// Mitsubishi GX Works2 project: pr2   PLC: Q03UDV

PROGRAM MAIN
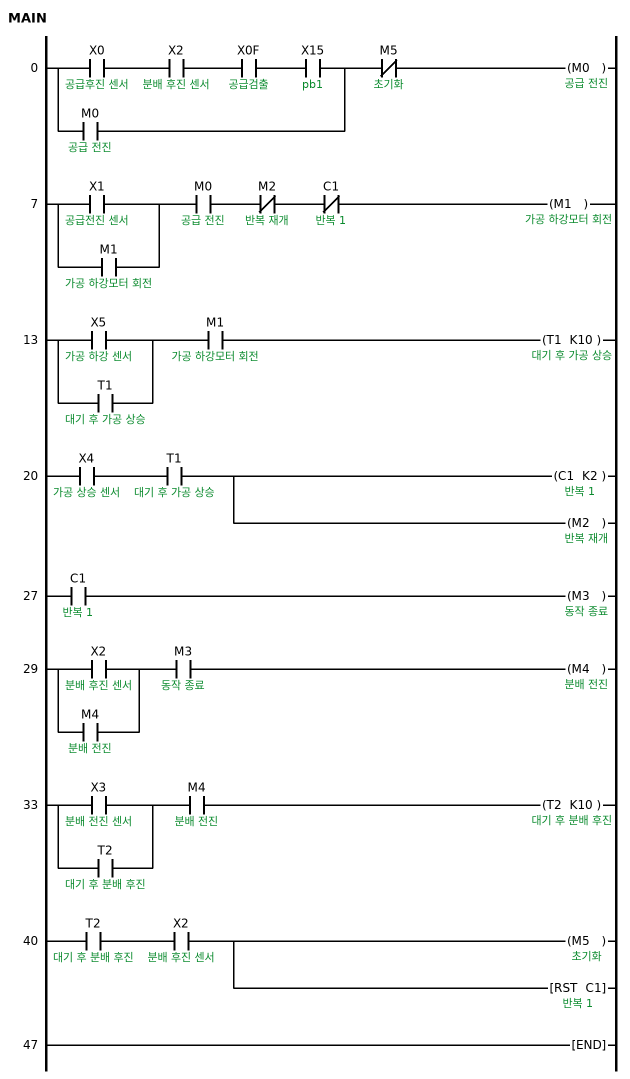
0     LD      X0  ; 공급후진 센서
      AND     X2  ; 분배 후진 센서
      AND     X0F  ; 공급검출
      AND     X15  ; pb1
      OR      M0  ; 공급 전진
      ANI     M5  ; 초기화
      OUT     M0  ; 공급 전진
7     LD      X1  ; 공급전진 센서
      OR      M1  ; 가공 하강모터 회전
      AND     M0  ; 공급 전진
      ANI     M2  ; 반복 재개
      ANI     C1  ; 반복 1
      OUT     M1  ; 가공 하강모터 회전
13    LD      X5  ; 가공 하강 센서
      OR      T1  ; 대기 후 가공 상승
      AND     M1  ; 가공 하강모터 회전
      OUT     T1 K10  ; 대기 후 가공 상승
20    LD      X4  ; 가공 상승 센서
      AND     T1  ; 대기 후 가공 상승
      OUT     C1 K2  ; 반복 1
      OUT     M2  ; 반복 재개
27    LD      C1  ; 반복 1
      OUT     M3  ; 동작 종료
29    LD      X2  ; 분배 후진 센서
      OR      M4  ; 분배 전진
      AND     M3  ; 동작 종료
      OUT     M4  ; 분배 전진
33    LD      X3  ; 분배 전진 센서
      OR      T2  ; 대기 후 분배 후진
      AND     M4  ; 분배 전진
      OUT     T2 K10  ; 대기 후 분배 후진
40    LD      T2  ; 대기 후 분배 후진
      AND     X2  ; 분배 후진 센서
      OUT     M5  ; 초기화
      RST     C1  ; 반복 1
47    END
END_PROGRAM

PROGRAM OUTPUT
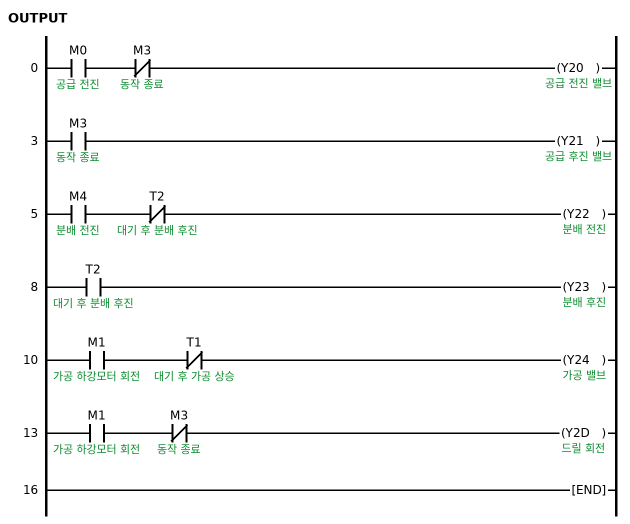
0     LD      M0  ; 공급 전진
      ANI     M3  ; 동작 종료
      OUT     Y20  ; 공급 전진 밸브
3     LD      M3  ; 동작 종료
      OUT     Y21  ; 공급 후진 밸브
5     LD      M4  ; 분배 전진
      ANI     T2  ; 대기 후 분배 후진
      OUT     Y22  ; 분배 전진
8     LD      T2  ; 대기 후 분배 후진
      OUT     Y23  ; 분배 후진
10    LD      M1  ; 가공 하강모터 회전
      ANI     T1  ; 대기 후 가공 상승
      OUT     Y24  ; 가공 밸브
13    LD      M1  ; 가공 하강모터 회전
      ANI     M3  ; 동작 종료
      OUT     Y2D  ; 드릴 회전
16    END
END_PROGRAM

// device comments not shown above
X6  ; 가공 하강 센서
